{attribute 'GeneratedUsingTerminal: EP7041-0002-0018'}
{attribute addProperty BoxType "EP7041-0002-0018"}
{attribute addProperty Id "AdsAddrAT %I*AMSADDR8Chn0AT %I*USINT1Chn1AT %I*USINT1StateAT %I*UINT2"}
{attribute addProperty CRC "1698221919"}
{attribute addProperty Size "12"}
TYPE InfoData_6538CF5F EXTENDS InputBase_8311D824 :
STRUCT
	{attribute addProperty Name "AdsAddr"}
	AdsAddr AT %I* : AMSADDR;
	{attribute addProperty Name "Chn0"}
	Chn0 AT %I* : USINT;
	{attribute addProperty Name "Chn1"}
	Chn1 AT %I* : USINT;
	{attribute addProperty Name "State"}
	State AT %I* : UINT;
END_STRUCT
END_TYPE

(* stored: Version 1.2.0.0, ProductVersion 3.1.4024.9
   DUT InfoData_6538CF5F: Id {7049319f-25b9-400b-a591-556139c43c02} *)
